		PreHtr_Proc							: REFERENCE TO BOOL							REF= PreHtr.Process.bActive;
		PreHtr_Val							: REFERENCE TO BOOL							REF= PreHtr.bActiveVal;
		PreHtr								: FB_ProcAggregateB							:= (iParent:=THIS^,					iLabel:=MyLabels.PreHtr,			Process:=(iLabel:=MyLabels.ProcPreRinse));
		Erc_Val								: REFERENCE TO BOOL							REF= Erc.bActiveVal;
		Erc									: FB_BA_AggregateB							:= (iParent:=THIS^,					iLabel:=MyLabels.Erc);
		Col_Val								: REFERENCE TO BOOL							REF= Col.bActiveVal;
		Col									: FB_BA_AggregateB							:= (iParent:=THIS^,					iLabel:=MyLabels.Col);
	{endregion}
	{region 'Plant'} 
		OpMode								: E_OpMod_AC								:= E_OpMod_AC.eOff;
		PlantCtrl_OpSta						: REFERENCE TO BOOL							REF= PlantCtrl.bOpSta;
		PlantCtrl_On						: REFERENCE TO BOOL							REF= PlantCtrl.bOn;
		PlantCtrl_PrVal						: REFERENCE TO UDINT						REF= PlantCtrl.nPresentValue;
		PlantCtrl_Step						: REFERENCE TO STRING						REF= PlantCtrl.sStep;
		PlantCtrl							: FB_BA_PlantCtrl := (
												iParent									:= THIS^,
												iLabel									:= MyLabels.PltCtrl,
												stOperation := (
													aOpMode								:= [ E_OpMod_AC.eDisturb,				E_OpMod_AC.eSmokeExtract,		E_OpMod_AC.eOff,			E_OpMod_AC.eOn,				E_OpMod_AC.eNightCool ],
													aPriority							:= [ E_BA_Priority.eCritical,			E_BA_Priority.eLifeSafety,		E_BA_Priority.eProgram,		E_BA_Priority.eProgram,		E_BA_Priority.eProgram ],
													aIgnoreFlags						:= [ E_BA_AggregateIgnoreFlags.Delay,	E_BA_AggregateIgnoreFlags.All,	0,							0,							0 ],
													aAggregates := [(
														iReference						:= DmprSu,
														aAggMode						:= [ 0,									100,							0,							100,						100 ]
													), (
														iReference						:= DmprEx,
														aAggMode						:= [ 0,									100,							0,							100,						100 ]
													), (
														iReference						:= PreHtr,
														aAggMode						:= [ E_OpMod_Binary.eOff,				E_OpMod_Binary.eOn,				E_OpMod_Binary.eOff,		E_OpMod_Binary.eOn,			E_OpMod_Binary.eOff ],
														bWaitForProcesses				:= TRUE
													), (
														iReference						:= Erc,
														aAggMode						:= [ E_OpMod_Binary.eOff,				E_OpMod_Binary.eOn,				E_OpMod_Binary.eOff,		E_OpMod_Binary.eOn,			E_OpMod_Binary.eOff ]
													), (
														iReference						:= Col,
														aAggMode						:= [ E_OpMod_Binary.eOff,				E_OpMod_Binary.eOn,				E_OpMod_Binary.eOff,		E_OpMod_Binary.eOn,			E_OpMod_Binary.eOff ]
													), (
														iReference						:= FanSu,
														aAggMode						:= [ E_OpMod_Step2.eOff,				E_OpMod_Step2.eStep2,			E_OpMod_Step2.eOff,			E_OpMod_Step2.eStep1,		E_OpMod_Step2.eStep2 ],
														tDelayStepDown					:= T#0S,
														tDelayStepUp					:= T#5S
													), (
														iReference						:= FanEx,
														aAggMode						:= [ E_OpMod_Step2.eOff,				E_OpMod_Step2.eStep2,			E_OpMod_Step2.eOff,			E_OpMod_Step2.eStep1,		E_OpMod_Step2.eStep2 ],
														tDelayStepDown					:= T#5S,
														tDelayStepUp					:= T#0S
													)]
											));
	{endregion}
END_VAR

SUPER^(); // FB_BA_View
DmprSu(); // FB_TimerAggregateA
FanSu(bEnCrit := NOT DmprSu.bOpen, nValCrit := E_OpMod_Step2.eOff); // FB_BA_AggregateM
DmprEx(); // FB_TimerAggregateA
FanEx(bEnCrit := NOT DmprEx.bOpen, nValCrit := E_OpMod_Step2.eOff); // FB_BA_AggregateM
PreHtr(); // FB_ProcAggregateB
Erc(); // FB_BA_AggregateB
Col(); // FB_BA_AggregateB
PlantCtrl(nOpMode := OpMode); // FB_BA_PlantCtrl

END_FUNCTION_BLOCK

// ---- SAMPLES/Demo/[Helper]/FunctionBlocks/Aggregates/FB_TimerAggregateA.TcPOU
// Some aggregate that has implemented a timer for demonstration.
FUNCTION_BLOCK FB_TimerAggregateA EXTENDS FB_BA_AggregateA
VAR_OUTPUT
	bOpen			: BOOL;
END_VAR
VAR
	Delay			: TON					:= (PT:=T#25S);
END_VAR

SUPER^();

Delay(IN := (bActiveEn AND (fActiveVal > 0.0)));
bOpen := Delay.Q;

END_FUNCTION_BLOCK

// ---- SAMPLES/Demo/[Helper]/FunctionBlocks/Aggregates/FB_ProcAggregateB.TcPOU
// Some aggregate that has implemented a process for demonstration.
FUNCTION_BLOCK FB_ProcAggregateB EXTENDS FB_BA_AggregateB
VAR
	Delay			: TON					:= (PT:=T#7S);
	Process			: FB_BA_Process			:= (iParent:=THIS^);
END_VAR

SUPER^();

Delay(IN := (bActiveEn AND bActiveVal));
Process(
	bEn := Delay.IN,
	bVal := (NOT Delay.Q)
);

END_FUNCTION_BLOCK

// ---- SAMPLES/Demo/Plant/FB_Plt_Init2.TcPOU
// How to initialize plant control with helper methods in "FB_init()".
// [Hint]
// > All reference-variables are implemented to ease monitoring of relevant variables.
FUNCTION_BLOCK FB_Plt_Init2 EXTENDS FB_BA_View
VAR
   	{region 'Aggregates'}
		DmprSu_Open							: REFERENCE TO BOOL							REF= DmprSu.bOpen;
		DmprSu_Val							: REFERENCE TO REAL							REF= DmprSu.fActiveVal;
		DmprSu								: FB_TimerAggregateA						:= (iParent:=THIS^,					iLabel:=MyLabels.DmprSu);
		FanSu_Val							: REFERENCE TO UDINT						REF= FanSu.nActiveVal;
		FanSu								: FB_BA_AggregateM							:= (iParent:=THIS^,					iLabel:=MyLabels.FanSu);
			 
		DmprEx_Open							: REFERENCE TO BOOL							REF= DmprEx.bOpen;
		DmprEx_Val							: REFERENCE TO REAL							REF= DmprEx.fActiveVal;
		DmprEx								: FB_TimerAggregateA						:= (iParent:=THIS^,					iLabel:=MyLabels.DmprEx);
		FanEx_Val							: REFERENCE TO UDINT						REF= FanEx.nActiveVal;
		FanEx								: FB_BA_AggregateM							:= (iParent:=THIS^,					iLabel:=MyLabels.FanEx);
			 
		PreHtr_Proc							: REFERENCE TO BOOL							REF= PreHtr.Process.bActive;
		PreHtr_Val							: REFERENCE TO BOOL							REF= PreHtr.bActiveVal;
		PreHtr								: FB_ProcAggregateB							:= (iParent:=THIS^,					iLabel:=MyLabels.PreHtr,			Process:=(iLabel:=MyLabels.ProcPreRinse));
		Erc_Val								: REFERENCE TO BOOL							REF= Erc.bActiveVal;
		Erc									: FB_BA_AggregateB							:= (iParent:=THIS^,					iLabel:=MyLabels.Erc);
		Col_Val								: REFERENCE TO BOOL							REF= Col.bActiveVal;
		Col									: FB_BA_AggregateB							:= (iParent:=THIS^,					iLabel:=MyLabels.Col);
	{endregion}
	{region 'Plant'} 
		OpMode								: E_OpMod_AC								:= E_OpMod_AC.eOff;
		PlantCtrl_OpSta						: REFERENCE TO BOOL							REF= PlantCtrl.bOpSta;
		PlantCtrl_On						: REFERENCE TO BOOL							REF= PlantCtrl.bOn;
		PlantCtrl_PrVal						: REFERENCE TO UDINT						REF= PlantCtrl.nPresentValue;
		PlantCtrl_Step						: REFERENCE TO STRING						REF= PlantCtrl.sStep;
		PlantCtrl							: FB_BA_PlantCtrl							:= (iParent:=THIS^,					iLabel:=MyLabels.PltCtrl);
	{endregion}
END_VAR

SUPER^(); // FB_BA_View
DmprSu(); // FB_TimerAggregateA
FanSu(bEnCrit := NOT DmprSu.bOpen, nValCrit := E_OpMod_Step2.eOff); // FB_BA_AggregateM
DmprEx(); // FB_TimerAggregateA
FanEx(bEnCrit := NOT DmprEx.bOpen, nValCrit := E_OpMod_Step2.eOff); // FB_BA_AggregateM
PreHtr(); // FB_ProcAggregateB
Erc(); // FB_BA_AggregateB
Col(); // FB_BA_AggregateB
PlantCtrl(nOpMode := OpMode); // FB_BA_PlantCtrl

METHOD FB_init : BOOL
VAR_INPUT
	bInitRetains : BOOL; // if TRUE, the retain variables are initialized (warm start / cold start)
	bInCopyCode : BOOL;  // if TRUE, the instance afterwards gets moved into the copy code (online change)
END_VAR
PlantCtrl.Clear();

// Add plant operations modes:
PlantCtrl.AddOperationMode(E_OpMod_AC.eDisturb,			E_BA_Priority.eCritical,	E_BA_AggregateIgnoreFlags.Delay);
PlantCtrl.AddOperationMode(E_OpMod_AC.eSmokeExtract,	E_BA_Priority.eLifeSafety,	E_BA_AggregateIgnoreFlags.All);
PlantCtrl.AddOperationMode(E_OpMod_AC.eOff,				E_BA_Priority.eProgram,		E_BA_AggregateIgnoreFlags.None);
PlantCtrl.AddOperationMode(E_OpMod_AC.eOn,				E_BA_Priority.eProgram,		E_BA_AggregateIgnoreFlags.None);
PlantCtrl.AddOperationMode(E_OpMod_AC.eNightCool,		E_BA_Priority.eProgram,		E_BA_AggregateIgnoreFlags.None);

// Add aggregates:
PlantCtrl.AddAggregate(DmprSu,	FALSE,	FALSE,	T#0S,	T#0S);
PlantCtrl.AddAggregate(DmprEx,	FALSE,	FALSE,	T#0S,	T#0S);
PlantCtrl.AddAggregate(PreHtr,	TRUE,	FALSE,	T#0S,	T#0S);
PlantCtrl.AddAggregate(Erc,		FALSE,	FALSE,	T#0S,	T#0S);
PlantCtrl.AddAggregate(Col,		FALSE,	FALSE,	T#0S,	T#0S);
PlantCtrl.AddAggregate(FanSu,	FALSE,	FALSE,	T#0S,	T#5S);
PlantCtrl.AddAggregate(FanEx,	FALSE,	FALSE,	T#5S,	T#0S);

// Apply aggregate operation modes dependant on corresponding plant operation modes:
PlantCtrl.AssignAggregate4x(E_OpMod_AC.eDisturb,		DmprSu, TO_UDINT(0),					FanSu, TO_UDINT(E_OpMod_Step2.eOff),		DmprEx, TO_UDINT(0),					FanEx, TO_UDINT(E_OpMod_Step2.eOff));
PlantCtrl.AssignAggregate4x(E_OpMod_AC.eSmokeExtract,	DmprSu, TO_UDINT(100),					FanSu, TO_UDINT(E_OpMod_Step2.eStep2),		DmprEx, TO_UDINT(100),					FanEx, TO_UDINT(E_OpMod_Step2.eStep2));
PlantCtrl.AssignAggregate4x(E_OpMod_AC.eOff,			DmprSu, TO_UDINT(0),					FanSu, TO_UDINT(E_OpMod_Step2.eOff),		DmprEx, TO_UDINT(0),					FanEx, TO_UDINT(E_OpMod_Step2.eOff));
PlantCtrl.AssignAggregate4x(E_OpMod_AC.eOn,				DmprSu, TO_UDINT(100),					FanSu, TO_UDINT(E_OpMod_Step2.eStep1),		DmprEx, TO_UDINT(100),					FanEx, TO_UDINT(E_OpMod_Step2.eStep1));
PlantCtrl.AssignAggregate4x(E_OpMod_AC.eNightCool,		DmprSu, TO_UDINT(100),					FanSu, TO_UDINT(E_OpMod_Step2.eStep2),		DmprEx, TO_UDINT(100),					FanEx, TO_UDINT(E_OpMod_Step2.eStep2));

PlantCtrl.AssignAggregate3x(E_OpMod_AC.eDisturb,		PreHtr, TO_UDINT(E_OpMod_Binary.eOff),	Erc, TO_UDINT(E_OpMod_Binary.eOff),			Col, TO_UDINT(E_OpMod_Binary.eOff));
PlantCtrl.AssignAggregate3x(E_OpMod_AC.eSmokeExtract,	PreHtr, TO_UDINT(E_OpMod_Binary.eOn),	Erc, TO_UDINT(E_OpMod_Binary.eOn),			Col, TO_UDINT(E_OpMod_Binary.eOn));
PlantCtrl.AssignAggregate3x(E_OpMod_AC.eOff,			PreHtr, TO_UDINT(E_OpMod_Binary.eOff),	Erc, TO_UDINT(E_OpMod_Binary.eOff),			Col, TO_UDINT(E_OpMod_Binary.eOff));
PlantCtrl.AssignAggregate3x(E_OpMod_AC.eOn,				PreHtr, TO_UDINT(E_OpMod_Binary.eOn),	Erc, TO_UDINT(E_OpMod_Binary.eOn),			Col, TO_UDINT(E_OpMod_Binary.eOn));
PlantCtrl.AssignAggregate3x(E_OpMod_AC.eNightCool,		PreHtr, TO_UDINT(E_OpMod_Binary.eOff),	Erc, TO_UDINT(E_OpMod_Binary.eOff),			Col, TO_UDINT(E_OpMod_Binary.eOff));
END_METHOD

END_FUNCTION_BLOCK

// ---- SAMPLES/Demo/Plant/FB_Plt_Init3.TcPOU
// How to initialize plant control with helper methods in "FB_init()".
// [Hint]
// > All reference-variables are implemented to ease monitoring of relevant variables.
FUNCTION_BLOCK FB_Plt_Init3 EXTENDS FB_BA_View
VAR
   	{region 'Aggregates'}
		DmprSu_Open							: REFERENCE TO BOOL							REF= DmprSu.bOpen;
		DmprSu_Val							: REFERENCE TO REAL							REF= DmprSu.fActiveVal;
		DmprSu								: FB_TimerAggregateA						:= (iParent:=THIS^,					iLabel:=MyLabels.DmprSu);
		FanSu_Val							: REFERENCE TO UDINT						REF= FanSu.nActiveVal;
		FanSu								: FB_BA_AggregateM							:= (iParent:=THIS^,					iLabel:=MyLabels.FanSu);
			 
		DmprEx_Open							: REFERENCE TO BOOL							REF= DmprEx.bOpen;
		DmprEx_Val							: REFERENCE TO REAL							REF= DmprEx.fActiveVal;
		DmprEx								: FB_TimerAggregateA						:= (iParent:=THIS^,					iLabel:=MyLabels.DmprEx);
		FanEx_Val							: REFERENCE TO UDINT						REF= FanEx.nActiveVal;
		FanEx								: FB_BA_AggregateM							:= (iParent:=THIS^,					iLabel:=MyLabels.FanEx);
			 
		PreHtr_Proc							: REFERENCE TO BOOL							REF= PreHtr.Process.bActive;
		PreHtr_Val							: REFERENCE TO BOOL							REF= PreHtr.bActiveVal;
		PreHtr								: FB_ProcAggregateB							:= (iParent:=THIS^,					iLabel:=MyLabels.PreHtr,			Process:=(iLabel:=MyLabels.ProcPreRinse));
		Erc_Val								: REFERENCE TO BOOL							REF= Erc.bActiveVal;
		Erc									: FB_BA_AggregateB							:= (iParent:=THIS^,					iLabel:=MyLabels.Erc);
		Col_Val								: REFERENCE TO BOOL							REF= Col.bActiveVal;
		Col									: FB_BA_AggregateB							:= (iParent:=THIS^,					iLabel:=MyLabels.Col);
	{endregion}
	{region 'Plant'} 
		OpMode								: E_OpMod_AC								:= E_OpMod_AC.eOff;
		PlantCtrl_OpSta						: REFERENCE TO BOOL							REF= PlantCtrl.bOpSta;
		PlantCtrl_On						: REFERENCE TO BOOL							REF= PlantCtrl.bOn;
		PlantCtrl_PrVal						: REFERENCE TO UDINT						REF= PlantCtrl.nPresentValue;
		PlantCtrl_Step						: REFERENCE TO STRING						REF= PlantCtrl.sStep;
		PlantCtrl							: FB_BA_PlantCtrl							:= (iParent:=THIS^,					iLabel:=MyLabels.PltCtrl);
	{endregion}
END_VAR

SUPER^(); // FB_BA_View
DmprSu(); // FB_TimerAggregateA
FanSu(bEnCrit := NOT DmprSu.bOpen, nValCrit := E_OpMod_Step2.eOff); // FB_BA_AggregateM
DmprEx(); // FB_TimerAggregateA
FanEx(bEnCrit := NOT DmprEx.bOpen, nValCrit := E_OpMod_Step2.eOff); // FB_BA_AggregateM
PreHtr(); // FB_ProcAggregateB
Erc(); // FB_BA_AggregateB
Col(); // FB_BA_AggregateB
PlantCtrl(nOpMode := OpMode); // FB_BA_PlantCtrl

METHOD FB_init : BOOL
VAR_INPUT
	bInitRetains : BOOL; // if TRUE, the retain variables are initialized (warm start / cold start)
	bInCopyCode : BOOL;  // if TRUE, the instance afterwards gets moved into the copy code (online change)
END_VAR
PlantCtrl.Clear();

// Add plant operations modes:
PlantCtrl.AddOperationMode(E_OpMod_AC.eDisturb,			E_BA_Priority.eCritical,	E_BA_AggregateIgnoreFlags.Delay);
PlantCtrl.AddOperationMode(E_OpMod_AC.eSmokeExtract,	E_BA_Priority.eLifeSafety,	E_BA_AggregateIgnoreFlags.All);
PlantCtrl.AddOperationMode(E_OpMod_AC.eOff,				E_BA_Priority.eProgram,		E_BA_AggregateIgnoreFlags.None);
PlantCtrl.AddOperationMode(E_OpMod_AC.eOn,				E_BA_Priority.eProgram,		E_BA_AggregateIgnoreFlags.None);
PlantCtrl.AddOperationMode(E_OpMod_AC.eNightCool,		E_BA_Priority.eProgram,		E_BA_AggregateIgnoreFlags.None);

// Add aggregates:
PlantCtrl.AddAggregate(DmprSu,	FALSE,	FALSE,	T#0S,	T#0S);
PlantCtrl.AddAggregate(DmprEx,	FALSE,	FALSE,	T#0S,	T#0S);
PlantCtrl.AddAggregate(PreHtr,	TRUE,	FALSE,	T#0S,	T#0S);
PlantCtrl.AddAggregate(Erc,		FALSE,	FALSE,	T#0S,	T#0S);
PlantCtrl.AddAggregate(Col,		FALSE,	FALSE,	T#0S,	T#0S);
PlantCtrl.AddAggregate(FanSu,	FALSE,	FALSE,	T#0S,	T#5S);
PlantCtrl.AddAggregate(FanEx,	FALSE,	FALSE,	T#5S,	T#0S);

// Apply aggregate operation modes dependant on corresponding plant operation modes:
PlantCtrl.AssignAggregate4x(E_OpMod_AC.eDisturb,		DmprSu, TO_UDINT(0),					FanSu, TO_UDINT(E_OpMod_Step2.eOff),		DmprEx, TO_UDINT(0),					FanEx, TO_UDINT(E_OpMod_Step2.eOff));
PlantCtrl.AssignAggregate4x(E_OpMod_AC.eSmokeExtract,	DmprSu, TO_UDINT(100),					FanSu, TO_UDINT(E_OpMod_Step2.eStep2),		DmprEx, TO_UDINT(100),					FanEx, TO_UDINT(E_OpMod_Step2.eStep2));
PlantCtrl.AssignAggregate4x(E_OpMod_AC.eOff,			DmprSu, TO_UDINT(0),					FanSu, TO_UDINT(E_OpMod_Step2.eOff),		DmprEx, TO_UDINT(0),					FanEx, TO_UDINT(E_OpMod_Step2.eOff));
PlantCtrl.AssignAggregate4x(E_OpMod_AC.eOn,				DmprSu, TO_UDINT(100),					FanSu, TO_UDINT(E_OpMod_Step2.eStep1),		DmprEx, TO_UDINT(100),					FanEx, TO_UDINT(E_OpMod_Step2.eStep1));
PlantCtrl.AssignAggregate4x(E_OpMod_AC.eNightCool,		DmprSu, TO_UDINT(100),					FanSu, TO_UDINT(E_OpMod_Step2.eStep2),		DmprEx, TO_UDINT(100),					FanEx, TO_UDINT(E_OpMod_Step2.eStep2));

PlantCtrl.AssignAggregate3x(E_OpMod_AC.eDisturb,		PreHtr, TO_UDINT(E_OpMod_Binary.eOff),	Erc, TO_UDINT(E_OpMod_Binary.eOff),			Col, TO_UDINT(E_OpMod_Binary.eOff));
PlantCtrl.AssignAggregate3x(E_OpMod_AC.eSmokeExtract,	PreHtr, TO_UDINT(E_OpMod_Binary.eOn),	Erc, TO_UDINT(E_OpMod_Binary.eOn),			Col, TO_UDINT(E_OpMod_Binary.eOn));
PlantCtrl.AssignAggregate3x(E_OpMod_AC.eOff,			PreHtr, TO_UDINT(E_OpMod_Binary.eOff),	Erc, TO_UDINT(E_OpMod_Binary.eOff),			Col, TO_UDINT(E_OpMod_Binary.eOff));
PlantCtrl.AssignAggregate3x(E_OpMod_AC.eOn,				PreHtr, TO_UDINT(E_OpMod_Binary.eOn),	Erc, TO_UDINT(E_OpMod_Binary.eOn),			Col, TO_UDINT(E_OpMod_Binary.eOn));
PlantCtrl.AssignAggregate3x(E_OpMod_AC.eNightCool,		PreHtr, TO_UDINT(E_OpMod_Binary.eOff),	Erc, TO_UDINT(E_OpMod_Binary.eOff),			Col, TO_UDINT(E_OpMod_Binary.eOff));
END_METHOD

END_FUNCTION_BLOCK

// ---- SAMPLES/Demo/Other/FB_Misc.TcPOU
// Miscellaneous.
FUNCTION_BLOCK FB_Misc EXTENDS FB_BA_View
VAR	
	// Intention:		Initialize some special UTF-8 characters.
	SpecialUtf8			: FB_BA_AV_Op := (
							iParent					:= THIS^,
							sDescription			:= wsLiteral_TO_UTF8("{äöüßéèêµ€° Ἀθῆναι İstanbul Київ}"),
							eUnit					:= E_BA_Unit.eOther_Percent,
							fValueRm				:= 5
						);
END_VAR

SUPER^();

SpecialUtf8();

END_FUNCTION_BLOCK

// ---- SAMPLES/Templates/Standard/POUs/Trade/General/EventClasses/FB_BA_EC01.TcPOU
// Template of event classes.
FUNCTION_BLOCK FB_BA_EC01 EXTENDS FB_BA_View
VAR CONSTANT
	OBJECT_NAME			: STRING					:= 'EC[InstID]';
END_VAR
VAR
	{region 'Alarm'}
		AlmSmpl			: FB_BA_EC := (
							iParent					:= THIS^,
							nInstanceID				:= 12,
							sObjectName				:= OBJECT_NAME,
							sDescription			:= '[Alarm (Einfach)]',
							eEventType				:= E_BA_EventType.eAlarm,
							eAlarmMode				:= E_BA_AlarmMode.eSimple,
							aPriority				:= [ 10, 11, 12 ]
						);
		AlmStd			: FB_BA_EC := (
							iParent					:= THIS^,
							nInstanceID				:= 11,
							sObjectName				:= OBJECT_NAME,
							sDescription			:= '[Alarm (Standard)]',
							eEventType				:= E_BA_EventType.eAlarm,
							eAlarmMode				:= E_BA_AlarmMode.eStandard,
							aPriority				:= [ 13, 14, 15 ]
						);
		AlmExt			: FB_BA_EC := (
							iParent					:= THIS^,
							nInstanceID				:= 10,
							sObjectName				:= OBJECT_NAME,
							sDescription			:= '[Alarm (Erweitert)]',
							eEventType				:= E_BA_EventType.eAlarm,
							eAlarmMode				:= E_BA_AlarmMode.eExtended,
							aPriority				:= [ 16, 17, 18 ]
						);
	{endregion}
	{region 'Disturb'}
		DstSmpl			: FB_BA_EC	:= (
							iParent					:= THIS^,
							nInstanceID				:= 52,
							sObjectName				:= OBJECT_NAME,
							sDescription			:= '[Störung (Einfach)]',
							eEventType				:= E_BA_EventType.eDisturb,
							eAlarmMode				:= E_BA_AlarmMode.eSimple,
							aPriority				:= [ 50, 51, 52 ]
						);
		DstStd			: FB_BA_EC := (
							iParent					:= THIS^,
							nInstanceID				:= 51,
							sObjectName				:= OBJECT_NAME,
							sDescription			:= '[Störung (Standard)]',
							eEventType				:= E_BA_EventType.eDisturb,
							eAlarmMode				:= E_BA_AlarmMode.eStandard,
							aPriority				:= [ 53, 54, 55 ]
						);
		DstExt			: FB_BA_EC := (
							iParent					:= THIS^,
							nInstanceID				:= 50,
							sObjectName				:= OBJECT_NAME,
							sDescription			:= '[Störung (Erweitert)]',
							eEventType				:= E_BA_EventType.eDisturb,
							eAlarmMode				:= E_BA_AlarmMode.eExtended,
							aPriority				:= [ 56, 57, 58 ]
						);
	{endregion}
	{region 'Maintenance'}
		MntnSmpl		: FB_BA_EC := (
							iParent					:= THIS^,
							nInstanceID				:= 92,
							sObjectName				:= OBJECT_NAME,
							sDescription			:= '[Wartung (Einfach)]',
							eEventType				:= E_BA_EventType.eMaintenance,
							eAlarmMode				:= E_BA_AlarmMode.eSimple,
							aPriority				:= [ 90, 91, 92 ]
						);
		MntnStd			: FB_BA_EC := (
							iParent					:= THIS^,
							nInstanceID				:= 91,
							sObjectName				:= OBJECT_NAME,
							sDescription			:= '[Wartung (Standard)]',
							eEventType				:= E_BA_EventType.eMaintenance,
							eAlarmMode				:= E_BA_AlarmMode.eStandard,
							aPriority				:= [ 93, 94, 95 ]
						);

		MntnExt			: FB_BA_EC := (
							iParent					:= THIS^,
							nInstanceID				:= 90,
							sObjectName				:= OBJECT_NAME,
							sDescription			:= '[Wartung (Erweitert)]',
							eEventType				:= E_BA_EventType.eMaintenance,
							eAlarmMode				:= E_BA_AlarmMode.eExtended,
							aPriority				:= [ 96, 97, 98 ]
						);
	{endregion}
	{region 'Notification'}
		NtfSmpl			: FB_BA_EC := (
							iParent					:= THIS^,
							nInstanceID				:= 132,
							sObjectName				:= OBJECT_NAME,
							sDescription			:= '[Benachrichtigung (Einfach)]',
							eEventType				:= E_BA_EventType.eNotification,
							eAlarmMode				:= E_BA_AlarmMode.eSimple,
							aPriority				:= [ 130, 131, 132 ]
						);
		NtfStd			: FB_BA_EC := (
							iParent					:= THIS^,
							nInstanceID				:= 131,
							sObjectName				:= OBJECT_NAME,
							sDescription			:= '[Benachrichtigung (Standard)]',
							eEventType				:= E_BA_EventType.eNotification,
							eAlarmMode				:= E_BA_AlarmMode.eStandard,
							aPriority				:= [ 133, 134, 135 ]
						);
	{endregion}
	{region 'Other'}
		OthSmpl			: FB_BA_EC := (
							iParent					:= THIS^,
							nInstanceID				:= 182,
							sObjectName				:= OBJECT_NAME,
							sDescription			:= '[Sonstiges (Einfach)]',
							eEventType				:= E_BA_EventType.eOther,
							eAlarmMode				:= E_BA_AlarmMode.eSimple,
							aPriority				:= [ 180, 181, 182 ]
						);
		OthStd			: FB_BA_EC := (
							iParent					:= THIS^,
							nInstanceID				:= 181,
							sObjectName				:= OBJECT_NAME,
							sDescription			:= '[Sonstiges (Standard)]',
							eEventType				:= E_BA_EventType.eOther,
							eAlarmMode				:= E_BA_AlarmMode.eStandard,
							aPriority				:= [ 183, 184, 185 ]
						);
	{endregion}
END_VAR

SUPER^(); // FB_BA_View
AlmSmpl(); // FB_BA_EC
AlmStd(); // FB_BA_EC
AlmExt(); // FB_BA_EC
DstSmpl(); // FB_BA_EC
DstStd(); // FB_BA_EC
DstExt(); // FB_BA_EC
MntnSmpl(); // FB_BA_EC
MntnStd(); // FB_BA_EC
MntnExt(); // FB_BA_EC
NtfSmpl(); // FB_BA_EC
NtfStd(); // FB_BA_EC
OthSmpl(); // FB_BA_EC
OthStd(); // FB_BA_EC

END_FUNCTION_BLOCK

// ---- SAMPLES/Demo/Optional Extensions/MAIN_OPTEXT.TcPOU
// Optional extensions.
// [Hint]
// - To stay maintainable and sustain a nice project overview it is recommended to declare these tools in your MAIN program.
PROGRAM MAIN_OPTEXT
VAR
	{region 'Settings'}
		// Intention:		Adjust certain ("BA_Param" related) settings via PLC code.
		//					> Feel free to implement as much instances as needed, where ever needed.
		Parameters			: FB_BA_Param := (
								EventEn_Simple			:= F_BA_EventTransition(TRUE, FALSE, FALSE),
								EventEn_Standard		:= F_BA_EventTransition(TRUE, FALSE, FALSE),
								EventEn_Extended		:= F_BA_EventTransition(TRUE, FALSE, TRUE),
								EvtMgmt_AckMode			:= E_BA_AcknowledgeMode.eEntire,
								
								// Intention:			Adjust access to some specific parameters (Leaving rest untouched).
								DefWriteAccess			:= F_BA_ParameterRolesBuilder()
															.Set(E_BA_Parameter.eEventEnable, E_BA_Role.eInternal)
															.Build()
							);

		// Intention:		Generically subscribe to certain events.
		//					> Use carefully (Refer to documentation - event subscribers are powerfull!)
		Events_LocObj		: FB_MyLocalObjectEvents;
	{endregion}
END_VAR

END_PROGRAM

// ---- SAMPLES/Demo/Optional Extensions/Events/FB_MyLocalObjectEvents.TcPOU
FUNCTION_BLOCK FB_MyLocalObjectEvents EXTENDS FB_BA_LocalObjectEventSubscriber

METHOD PRIVATE IsPressure : BOOL
VAR_INPUT
	eUnit		: E_BA_Unit;
END_VAR
IsPressure := (E_BA_Unit.ePressure_Pascals <= eUnit) AND_THEN (eUnit <= E_BA_Unit.ePressure_InchesOfMercury);
END_METHOD

METHOD PRIVATE IsTemperature : BOOL
VAR_INPUT
	eUnit		: E_BA_Unit;
END_VAR
IsTemperature := (E_BA_Unit.eTemperature_DegreesCelsius <= eUnit) AND_THEN (eUnit <= E_BA_Unit.eTemperature_DegreeDaysFahrenheit);
END_METHOD

METHOD PROTECTED OnInitInstanceId
VAR_INPUT
	iObject			: I_BA_Object;
END_VAR
VAR_INST
	_nID_Temp		: UDINT						:= 5000;				// First ID to assign to temperature sensors.
	_nID_Prs		: UDINT						:= 6000;				// First ID to assign to pressure sensors.
END_VAR
VAR
	_iAnalogObj		: I_BA_AnalogObject;
	_nID			: REFERENCE TO UDINT;
END_VAR
// Sample 1) Generate instance ID related to configured units.

IF (iObject.InstanceID <> 0) THEN
	; // ID already assigned.
ELSIF (iObject.DataClass <> E_BA_DataClass.eAnalog) THEN
	; // Skip.
ELSIF (NOT __QUERYINTERFACE(iObject, _iAnalogObj)) THEN
	; // Failed to convert interface.
ELSE
	// Determine range of instance IDs:
	IF (IsTemperature(_iAnalogObj.Unit)) THEN
		_nID REF= _nID_Temp;
	ELSIF (IsPressure(_iAnalogObj.Unit)) THEN
		_nID REF= _nID_Prs;
	ELSE
		RETURN; // Skip (Instance ID will be auto-generated).
	END_IF
		
	// Assign instance ID:
	_iAnalogObj.InstanceID := _nID;
	iObject.LogMsg.Show1(ADSLOG_MSGTYPE_HINT, 'OIII21', 'Assigned instance ID %d.', F_UDINT(_nID), FALSE);
	
	_nID := (_nID+1);
END_IF
END_METHOD

METHOD PROTECTED OnProjectStateChanged
VAR_INPUT
	eState			: E_BA_ProjectState;
END_VAR
// Sample 1) Evaluate project state.
CASE (eState) OF
	E_BA_ProjectState.eFirstOpCycle:
		F_BA_LogMessage(ADSLOG_MSGTYPE_HINT, 'OPSC04', 'Initialization done: project is operational.');
	
	E_BA_ProjectState.Error:
		F_BA_LogMessage(ADSLOG_MSGTYPE_HINT, 'OPSC07', 'Initialization failed!');
	
END_CASE
END_METHOD

END_FUNCTION_BLOCK
